# B&R Automation Studio project AriesV2 (part 3)

### bgsscanf.c
```c
#ifndef _BG_SSCANF_C
#define _BG_SSCANF_C
/*
Source:
http://www.koders.com/c/fid1D51E1E6F4F922088DF508FFEEEEC702AFED6333.aspx?s=__v_scanf
*/

//#include <stdarg.h>
//#include <limits.h>
//#include <string.h>

#define GBLONG_MAX 2147483647L
#define GBLONG_MIN (-GBLONG_MAX-1)
#define GBULONG_MAX (GBLONG_MAX * 2UL + 1)

extern long int strtol ( const char * str, char ** endptr, int base );

#define WANT_FLOATING_POINT_IN_SCANF 1
#define WANT_CHARACTER_CLASSES_IN_SCANF 1

#define	EOF	(-1)

struct arg_scanf {
  void *data;
  int (*getch)(void*);
  int (*putch)(int,void*);
};

struct str_data {
  unsigned char* str;
};

static int sgetc(struct str_data* sd) {
  register unsigned int ret = *(sd->str++);
  return (ret)?(int)ret:-1;
}

static int sputc(int c, struct str_data* sd) {
  return (*(--sd->str)==c)?c:-1;
}

#define A_GETC(fn)	(++consumed,(fn)->getch((fn)->data))
#define A_PUTC(c,fn)	(--consumed,(fn)->putch((c),(fn)->data))

static int isspace(int c)
{
	return ((c==(int)' ')) ? 1 : 0;
}

static int isdigit(int c)
{
	return ((c>=(int)'0') && (c<=(int)'9')) ? 1 : 0;
}

int __v_scanf(struct arg_scanf* fn, const unsigned char *format, va_list arg_ptr)
{
  unsigned int ch;	/* format act. char */
  int n=0;

  /* arg_ptr tmps */
#ifdef WANT_FLOATING_POINT_IN_SCANF
  double *pd;
  float  *pf;
#endif
  long   *pl;
  short  *ph;
  int    *pi;
  char    *s;

  unsigned int consumed=0;

  /* get one char */
  int tpch= A_GETC(fn);

  while (*format)
  {
    ch=*format++;
    switch (ch) {
    /* end of format string ?!? */
    case 0: return 0;

    /* skip spaces ... */
    case ' ':
    case '\f':
    case '\t':
    case '\v':
    case '\n':
    case '\r':
      while((*format)&&(isspace(*format))) ++format;
      while(isspace(tpch)) tpch=A_GETC(fn);
      break;

    /* format string ... */
    case '%':
      {
	unsigned int _div=0;
	int width=-1;
	char flag_width=0;
	char flag_discard=0;
	char flag_half=0;
	char flag_long=0;
	char flag_longlong=0;

in_scan:
	ch=*format++;
	if(ch!='n' && tpch==-1) goto err_out;
	switch (ch) {
	/* end of format string ?!? */
	case 0: return 0;

	/* check for % */
	case '%':
	  if ((unsigned char)tpch != ch) goto err_out;
	  tpch=A_GETC(fn);
	  break;

	/* FLAGS */
	case '*':
	  flag_discard=1;
	  goto in_scan;
	case 'h':
	  flag_half=1;
	  goto in_scan;
	case 'l':
	  if (flag_long) flag_longlong=1;
	  flag_long=1;
	  goto in_scan;
	case 'q':
	case 'L':
	  flag_longlong=1;
	  goto in_scan;

	/* WIDTH */
	case '0':
	case '1':
	case '2':
	case '3':
	case '4':
	case '5':
	case '6':
	case '7':
	case '8':
	case '9':
	  width=strtol((const char*)(format-1),&s,10);
	  format=(unsigned char*)s;
	  flag_width=1;
	  goto in_scan;

	/* scan for integer / strtol reimplementation ... */
	case 'p':
	case 'X':
	case 'x':
	  _div+=6;
	case 'd':
	  _div+=2;
	case 'o':
	  _div+=8;
	case 'u':
	case 'i':
	  {
	    unsigned long v=0;
	    unsigned int consumedsofar;
	    int neg=0;
	    while(isspace(tpch)) tpch=A_GETC(fn);
	    if (tpch=='-') {
	      tpch=A_GETC(fn);
	      neg=1;
	    }

	    if (tpch=='+') tpch=A_GETC(fn);

	    if (tpch==-1) return n;
	    consumedsofar=consumed;

	    if (!flag_width) {
	      if ((_div==16) && (tpch=='0')) goto scan_hex;
	      if (!_div) {
		_div=10;
		if (tpch=='0') {
		  _div=8;
scan_hex:
		  tpch=A_GETC(fn);
		  if ((tpch|32)=='x') {
		    tpch=A_GETC(fn);
		    _div=16;
		  }
		}
	      }
	    }
	    while ((width)&&(tpch!=-1)) {
	      register unsigned long c=tpch&0xff;
	      register unsigned long d=c|0x20;
	      c=(d>='a'?d-'a'+10:c<='9'?c-'0':0xff);
	      if (c>=_div) break;
	      d=v*_div;
	      v=(d<v)?GBULONG_MAX:d+c;
	      --width;
	      tpch=A_GETC(fn);
	    }

	    if (consumedsofar==consumed) return n;

	    if ((ch|0x20)<'p') {
	      register long l=v;
	      if (v>=-((unsigned long)GBLONG_MIN)) {
		l=(neg)?GBLONG_MIN:GBLONG_MAX;
	      }
	      else {
		if (neg) v*=-1;
	      }
	    }
	    if (!flag_discard) {
	      if (flag_long) {
		pl=(long *)va_arg(arg_ptr,long*);
		*pl=v;
	      } else if (flag_half) {
		ph=(short*)va_arg(arg_ptr,short*);
		*ph=v;
	      } else {
		pi=(int *)va_arg(arg_ptr,int*);
		*pi=v;
	      }
	      if(consumedsofar<consumed) ++n;
	    }
	  }
	  break;

	/* FIXME: return value of *scanf with ONE float maybe -1 instead of 0 */
#ifdef WANT_FLOATING_POINT_IN_SCANF
	/* floating point numbers */
	case 'e':
	case 'E':
	case 'f':
	case 'g':
	  {
	    double d=0.0;
	    int neg=0;
	    unsigned int consumedsofar;

	    while(isspace(tpch)) tpch=A_GETC(fn);

	    if (tpch=='-') {
	      tpch=A_GETC(fn);
	      neg=1;
	    }
	    if (tpch=='+') tpch=A_GETC(fn);

	    consumedsofar=consumed;

	    while (isdigit(tpch)) {
	      d=d*10+(tpch-'0');
	      tpch=A_GETC(fn);
	    }
	    if (tpch=='.') {
	      double factor=.1;
	      consumedsofar++;
	      tpch=A_GETC(fn);
	      while (isdigit(tpch)) {
		d=d+(factor*(tpch-'0'));
		factor/=10;
		tpch=A_GETC(fn);
	      }
	    }
	    if (consumedsofar==consumed) return n;	/* error */
	    if ((tpch|0x20)=='e') {
	      int exp=0, prec=tpch;
	      double factor=10;
	      tpch=A_GETC(fn);
	      if (tpch=='-') {
		factor=0.1;
		tpch=A_GETC(fn);
	      } else if (tpch=='+') {
		tpch=A_GETC(fn);
	      } else {
		d=0;
		if (tpch!=-1) A_PUTC(tpch,fn);
		tpch=prec;
		goto exp_out;
	      }
	      consumedsofar=consumed;
	      while (isdigit(tpch)) {
		exp=exp*10+(tpch-'0');
		tpch=A_GETC(fn);
	      }
	      if (consumedsofar==consumed) return n;	/* error */
	      while (exp) {	/* as in strtod: XXX: this introduces rounding errors */
		d*=factor; --exp;
	      }
	    }
exp_out:
	    if (!flag_discard) {
	      if (flag_long) {
		pd=(double *)va_arg(arg_ptr,double*);
		*pd=d;
	      } else {
		pf=(float *)va_arg(arg_ptr,float*);
		*pf=d;
	      }
	      ++n;
	    }
	  }
	  break;
#endif

	/* char-sequences */
	case 'c':
	  if (!flag_discard) {
	    s=(char *)va_arg(arg_ptr,char*);
	    ++n;
	  }
	  if (!flag_width) width=1;
	  while (width && (tpch!=-1)) {
	    if (!flag_discard) *(s++)=tpch;
	    --width;
	    tpch=A_GETC(fn);
	  }
	  break;

	/* string */
	case 's':
	  if (!flag_discard) s=(char *)va_arg(arg_ptr,char*);
	  while(isspace(tpch)) tpch=A_GETC(fn);
	  if (tpch==-1) break;		/* end of scan -> error */
	  while (width && (tpch!=-1) && (!isspace(tpch))) {
	    if (!flag_discard) *s=tpch;
	    if (tpch) ++s; else break;
	    --width;
	    tpch=A_GETC(fn);
	  }
	  if (!flag_discard) { *s=0; ++n; }
	  break;

	/* consumed-count */
	case 'n':
	  if (!flag_discard) {
	    pi=(int *)va_arg(arg_ptr,int *);
            *pi=consumed-1;
	  }
	  break;

#ifdef WANT_CHARACTER_CLASSES_IN_SCANF
	case '[':
	  {
	    char cset[256];
	    int flag_not=0;
	    int flag_dash=0;
	    memset(cset,0,sizeof(cset));
	    ch=*format++;
	    /* first char specials */
	    if (ch=='^') {
	      flag_not=1;
	      ch=*format++;
	    }
	    if ((ch=='-')||(ch==']')) {
	      cset[ch]=1;
	      ch=*format++;
	    }
	    /* almost all non special chars */
	    for (;(*format) && (*format!=']');++format) {
	      if (flag_dash) {
		register unsigned char tmp=*format;
		for (;ch<=tmp;++ch) cset[ch]=1;
		flag_dash=0;
		ch=*format;
	      }
	      else if (*format=='-') flag_dash=1;
	      else {
		cset[ch]=1;
		ch=*format;
	      }
	    }
	    /* last char specials */
	    if (flag_dash) cset['-']=1;
	    else cset[ch]=1;

	    /* like %c or %s */
	    if (!flag_discard) {
	      s=(char *)va_arg(arg_ptr,char*);
	      ++n;
	    }
	    while (width && (tpch>=0) && (cset[tpch]^flag_not)) {
	      if (!flag_discard) *s=tpch;
	      if (tpch) ++s; else break;
	      --width;
	      tpch=A_GETC(fn);
	    }
	    if (!flag_discard) *s=0;
	    ++format;
	  }
	  break;
#endif
	default:
	  goto err_out;
	}
      }
      break;

    /* check if equal format string... */
    default:
      if ((unsigned char)tpch != ch) goto err_out;
      tpch=A_GETC(fn);
      break;
    }
  }

  /* maybe a "%n" follows */
  if(*format) {
    while(isspace(*format)) format++;
    if(format[0] == '%' && format[1] == 'n') {
      pi = (int *) va_arg(arg_ptr, int *);
      *pi = consumed - 1;
    }
  }

err_out:
  if (tpch<0 && n==0) return EOF;
  A_PUTC(tpch,fn);
  return n;
}

int bgvsscanf(const char* str, const char* format, va_list arg_ptr)
{
  struct str_data  fdat = { (unsigned char*)str };
  struct arg_scanf farg = { (void*)&fdat, (int(*)(void*))sgetc, (int(*)(int,void*))sputc };
  return __v_scanf(&farg,format,arg_ptr);
}

int bgsscanf(const char *str, const char *format, ...)
{
  int n;
  va_list arg_ptr;
  va_start(arg_ptr, format);
  n=bgvsscanf(str,format,arg_ptr);
  va_end (arg_ptr);
  return n;
}

#endif
```

### bgTimer1ms.c
```c
/********************************************************************
 * COPYRIGHT -- belgor
 ********************************************************************
 * Package: bglib
 * File: bgTimer1ms.c
 * Author: goran
 * Created: October 05, 2011
 *******************************************************************/

#include <bur/plctypes.h>
#ifdef _DEFAULT_INCLUDES
	#include <AsDefault.h>
#endif

//#include <standard.h>

#ifndef _BG_TIMER_x1MS_C
#define _BG_TIMER_x1MS_C

void bgTimerExecute(TON_typ *timer){
	TON(timer);
}

void bgTimerStart(TON_typ *timer, int timeoutTime){
	timer->IN = 0;
	TON(timer);
	timer->IN = 1;
	timer->PT = timeoutTime;
	TON(timer );
}

void bgTimerStop(TON_typ *timer){
	timer->IN = 0;
	TON(timer);
}

BOOL  bgTimerIsTimeOut(TON_typ *timer){
	return timer->Q;
}

UDINT bgTimerTimeRemaining(TON_typ *timer){
	return (timer->PT - timer->ET);
}

UDINT bgTimerTimeElapsed( TON_typ *timer ) {
	return (timer->ET);
}

#endif //_BG_TIMER_x1MS_C
```

### HMI.typ
```iecst
(********************************************************************
 * COPYRIGHT -- piedmont
 ********************************************************************
 * Package: HMI
 * File: HMI.typ
 * Author: goran
 * Created: August 28, 2013
 ********************************************************************
 * Data types of package HMI
 ********************************************************************)
(*########################################################################*)
(*HMI key assinged PV-s (i.e. page navigation, save btns, etc)*)
(*########################################################################*)

TYPE
	hmiControlLogicKeys_typ : 	STRUCT
		btnRestartLoginTimer : USINT; (*1-means that login timer restart is requested*)
		btnLoginIcon : USINT; (*1-means that login logo (icon) is pressed*)
		menuKeyPressLT : ARRAY[0..HMI_ENUM_MENU_ITEMS_LT]OF BOOL; (*Mom keys connected to menu items LF*)
		menuKeyPressRT : ARRAY[0..HMI_ENUM_MENU_ITEMS_RT]OF BOOL; (*Mom keys connected to menu items RT*)
	END_STRUCT;
END_TYPE

(*########################################################################*)
(*HMI navigation PV-s (i.e. PV-s assigned to required VC PV-s such as currentPage, etc)*)
(*########################################################################*)

TYPE
	hmiNavigationLogic_typ : 	STRUCT
		changePage : USINT;
		currentPage : USINT;
		htmlCurrentURL : STRING[127];
		htmlChangeURL : STRING[127];
		currentPageText : STRING[31];
		prevPage : USINT;
		nextPage : USINT;
		pageInit : BOOL;
		pageExit : BOOL;
		state : USINT;
		currentStateText : STRING[31];
		statePrev : USINT;
		stateNext : USINT;
		loginLevel : UDINT;
		stateInit : BOOL;
		tmr1 : TON; (*Alert message control timer*)
		tmr2 : TON; (*Unack alarms message alert blinking timer*)
		tmr3 : TON; (*Password level reset timer*)
		tmr3RemainingTimeSec : UDINT;
		tmr3RemainingTimeMin : UDINT;
		tmr4 : TON;
	END_STRUCT;
END_TYPE

(*########################################################################*)
(*HMI related status control PV-s (i.e. visibility, locking, etc)*)
(*########################################################################*)

TYPE
	hmiControlLogicStatus_typ : 	STRUCT
		visibleSaveCfg : UINT;
		menuVisibleLT : UINT; (*Main menu LF visibility control *)
		menuVisibleRT : UINT; (*Main menu RT visibility control *)
		menuVisibleRTItems : ARRAY[0..HMI_ENUM_MENU_ITEMS_RT]OF UINT; (*Main menu items RT visibility control - for buttons stacked on top of each other in the upper, rt *)
		menuIndexLT : UINT; (*Main menu currently selected menu item - LF*)
		show_motion_tab : USINT;
		show_Aux_tab : USINT;
		show_io_tab : UINT;
		menuIndexRT : UINT; (*Main menu currently selected menu item - RT*)
		loginVisibleGE1 : USINT; (*Visibility control for login level related stuff - set to visible (0) if login level >= 1; othervise set to 1 (i.e. loginLevel < 1)*)
		loginVisibleGE2 : USINT; (*Visibility control for login level related stuff - set to visible (0) if login level >= 2; othervise set to 1 (i.e. loginLevel < 2)*)
		loginVisibleGE3 : USINT; (*Visibility control for login level related stuff - set to visible (0) if login level >= 2; othervise set to 1 (i.e. loginLevel < 2)*)
		menuLFHideTimer : TON; (*timer of automaticaly hiding LF dropdown menu*)
		menuRTHideTimer : TON; (*timer of automaticaly hiding RT dropdown menu*)
		tabKeysRadioDataPoint : USINT; (*DP that tab button are writing to in order to create radio buttons/tab view effect*)
		tabKeysRadioArray : ARRAY[0..HMI_ENUM_TAB_KEYS_MAX]OF USINT;
		tabKeysToggle : ARRAY[0..HMI_ENUM_MENU_ITEMS_LT]OF USINT;
		passwordStrings : ARRAY[0..HMI_PWD_LEVELS]OF STRING[HMI_PWD_MAXLEN]; (*Password strings used for loginLevel control*)
	END_STRUCT;
END_TYPE

(*=============================================================================*)
(*Recipe related HMI logic.*)
(*=============================================================================*)

TYPE
	hmiRecipeLogic_typ : 	STRUCT
		recVisible : USINT; (*Recipe related visibility control*)
		recSelectIdx : UINT; (*Recipe list index*)
		recSelectIdxMax : UINT; (*Recipe list index*)
		recSaveAsIdx : UINT; (*Recipe index for SaveAs action*)
		recSelectName : STRING[80]; (*Name of the currently selected recipe from the recipe list*)
		btnLockedActivate : USINT; (*Button lock control*)
		btnLockedNew : USINT; (*Button lock control*)
		btnLockedDelete : USINT; (*Button lock control*)
		btnLockedSaveAs : USINT; (*Button lock control*)
		btnActivate : BOOL; (*mom btn to Activate a recipe*)
		btnNew : BOOL; (*mom btn to New a recipe*)
		btnDelete : BOOL; (*mom btn to Delete a recipe*)
		btnSaveAs : BOOL; (*mom btn to SaveAs a recipe*)
		stateRecipes : UDINT;
	END_STRUCT;
END_TYPE

(*=============================================================================*)
(*Fileio Items*)
(*=============================================================================*)
(*=============================================================================*)
(*Tabs Control*)
(*=============================================================================*)
(*=============================================================================*)
(*HMI related navigation and control logic.*)
(*=============================================================================*)
(*Insert your comment here.*)
(*Insert your comment here.*)

TYPE
	hmiTableTrigger_typ : 	STRUCT
		Rec : BOOL;
		Cfg : BOOL;
	END_STRUCT;
	hmiTableLoad_typ : 	STRUCT
		Trigger : BOOL;
	END_STRUCT;
	hmiTables_typ : 	STRUCT
		Trigger : hmiTableTrigger_typ;
		Load : hmiTableLoad_typ;
	END_STRUCT;
END_TYPE

(*Insert your comment here.*)

TYPE
	hmiControlLogic_typ : 	STRUCT
		status : hmiControlLogicStatus_typ;
		keys : hmiControlLogicKeys_typ;
		prv : hmiNavigationLogic_typ; (*Hmi (panel) private data for handling screen navigation and hmi logic. Used only wihin HMI.*)
		recipes : hmiRecipeLogic_typ;
		alertMsg : hmiAlert_typ;
		dialogMsg : hmiDialog_typ;
		tables : hmiTables_typ;
	END_STRUCT;
END_TYPE
```

### HMI_Pages.typ
```iecst
TYPE
	HMI_Page_Enum :
		( (*IMPORTANTNOTE: if the application is going to work correctly, you have to MANUALLY ADD all of the enumerations below AND make sure they line up with the hmi page numbers. *)
		HMI_00_STARTUP := 0,
		HMI_HOME_10_DASHBOARD := 10,
		HMI_RECIPE_20_SELECT := 20,
		HMI_RECIPE_21_PVLIST := 21,
		HMI_CONFIG_30_SELECT := 30,
		HMI_CONFIG_31_PVLIST := 31,
		HMI_LOGIN_40_MAIN := 40,
		HMI_LOGIN_41_OPERATOR := 41,
		HMI_LOGIN_42_SETUP := 42,
		HMI_LOGIN_43_ENGINEER := 43,
		HMI_LOGIN_44_HERNON := 44,
		HMI_LOGIN_45_FACTORY := 45,
		HMI_DIAGNOSTICS_50_ALARMS := 50,
		HMI_DIAGNOSTICS_51_ALRMHST := 51,
		HMI_DIAGNOSTICS_52_SDM := 52,
		HMI_DIAGNOSTICS_53_SYSLOG := 53,
		HMI_MOTION_60_IO_DISPENSE := 60,
		HMI_MOTION_61_IO_MOTORS := 61,
		HMI_MOTION_62_DISPENSE_TREND := 62,
		HMI_MOTION_63_IO_INSPECT_IO := 63,
		HMI_MOTION_64_IO_INSPECT_TREND := 64,
		HMI_MOTION_65_IO_LOADER := 65,
		HMI_MOTION_66_IO_SAFETY := 66,
		HMI_MOTION_67_IO_ETC := 67,
		HMI_MOTION_68_IO_SENSOR := 68,
		HMI_MOTION_69_IO_LOAD5215 := 69,
		HMI_ACP_70_AXIS_OVERVIEW := 70,
		HMI_ACP_71_AXIS_REF := 71,
		HMI_ACP_72_AXIS_MOVE := 72,
		HMI_ACP_73_AXIS_SETUP := 73,
		HMI_ACP_74_CAM_CTRL := 74,
		HMI_ACP_75_CAM_SETUP := 75,
		HMI_ACP_76_CAM_TRACE := 76,
		HMI_AUX_90_FILE := 90
		);
END_TYPE
```

### HMIdialog.typ
```iecst
(********************************************************************
 * COPYRIGHT -- piedmont
 ********************************************************************
 * Package: HMI
 * File: HMI.typ
 * Author: goran
 * Created: August 28, 2013
 ********************************************************************
 * Data types of package HMI
 ********************************************************************)
(*########################################################################*)
(*HMI object - DIALOG (OK, Cancel)*)
(*########################################################################*)

TYPE
	hmiDialog_typ : 	STRUCT
		message : STRING[512];
		result : UINT; (*value returned when button pressed (0-busy, button not pressed, dialog active, OK pressed returns resultForOk (eg.1); Cancel pressed returns resultForCancel (eg.2)*)
		resultForOk : UINT; (*value to return when Ok pressed (if 0 return value is 1)*)
		resultForCancel : UINT; (*value to return when Cancel pressed (if 0 return value is 2)*)
		timeoutConfig : UINT; (*configuration input that defines meaning of the timeout. If 0 > timeout means cancel; if 1> timeout means ok*)
		status : UINT; (*Status for common dialog layer*)
		tmr1RemainingTimeSec : UDINT; (*Timer remaining time (sec)*)
		btnOk : UINT; (*press on button OK sets this value to 1*)
		btnCancel : UINT; (*press on button Cancel sets this value to 1*)
		tmr1 : TON; (*Dialog control timer*)
	END_STRUCT;
END_TYPE
```

### Program Logical/HMI/HMI_Alarms

#### Variables.var
```iecst
VAR
	ii_alarms : UDINT;
	tmp_alarm_counter : UDINT;
END_VAR
```

#### Cyclic.st
```iecst
PROGRAM _CYCLIC
	brsmemcpy(ADR(AppAlarms.AlarmImage[0]), 	ADR(gAlarms), 					SIZEOF(Machine_Alarms_typ));

	brsmemcpy(ADR(gAcknowledge), 				ADR(AppAlarms.AlarmImage[0]), 	SIZEOF(Machine_Alarms_typ));

//	tmp_alarm_counter := 0;
//
//	FOR ii_alarms := 0 TO MAX_IDX_ALARMS BY 1 DO
//		IF gMachine.HMI.AlarmControls.Dispense.AlarmImage[ii_alarms] THEN
//			tmp_alarm_counter := tmp_alarm_counter + 1;
//		END_IF;
//
//		IF gMachine.HMI.AlarmControls.Inspect.AlarmImage[ii_alarms] THEN
//			tmp_alarm_counter := tmp_alarm_counter + 1;
//		END_IF;
//
//		IF gMachine.HMI.AlarmControls.Sensor.AlarmImage[ii_alarms] THEN
//			tmp_alarm_counter := tmp_alarm_counter + 1;
//		END_IF;
//
//		IF gMachine.HMI.AlarmControls.Safety.AlarmImage[ii_alarms] THEN
//			tmp_alarm_counter := tmp_alarm_counter + 1;
//		END_IF;
//
//		IF gMachine.HMI.AlarmControls.RecCfg.AlarmImage[ii_alarms] THEN
//			tmp_alarm_counter := tmp_alarm_counter + 1;
//		END_IF;
//
//		IF gMachine.HMI.AlarmControls.Hardware.AlarmImage[ii_alarms] THEN
//			tmp_alarm_counter := tmp_alarm_counter + 1;
//		END_IF;
//
//		IF gMachine.HMI.AlarmControls.Motor.AlarmImage[ii_alarms] THEN
//			tmp_alarm_counter := tmp_alarm_counter + 1;
//		END_IF;
//	END_FOR;

	IF gAlarmResetRequested THEN
		brsmemset(ADR(gAlarms), 0, 		SIZEOF(Machine_Alarms_typ));

		gAlarmResetRequested := FALSE;
	END_IF;
//
//	IF Alarm_Control.ActiveAlarms = 0 AND Alarm_Control.PendingAlarms = 0 AND tmp_alarm_counter = 0 THEN
//		gAlarmState := 0;
//	ELSIF Alarm_Control.ActiveAlarms = 0 AND Alarm_Control.PendingAlarms = 0 AND tmp_alarm_counter > 0 THEN
//		gAlarmState := 1;
//	ELSIF Alarm_Control.ActiveAlarms = 0 AND Alarm_Control.PendingAlarms > 0 THEN
//		gAlarmState := 2;
//	ELSE
//		gAlarmState := 3;
//	END_IF;

	AppAlarms_FBK();
//
//	gMachine.HMI.Dashboard.Application_Errors_Active := tmp_alarm_counter;
//	gMachine.HMI.Dashboard.System_Alarms_Active := Alarm_Control.ActiveAlarms;
//	gMachine.HMI.Dashboard.System_Alarms_Pending := Alarm_Control.PendingAlarms;
END_PROGRAM
```

### Program Logical/HMI/hmilogic

#### hmiDialog.h
```c
/********************************************************************
 * COPYRIGHT -- piedmont
 ********************************************************************
 * Program: hmilogic
 * File: hmiDialog.h
 * Author: goran
 * Created: September 05, 2013
 *******************************************************************/

#include <bur/plctypes.h>
#ifdef _DEFAULT_INCLUDES
#include <AsDefault.h>
#endif
BOOL hmiDialogIsActive(hmiDialog_typ* p);
void hmiDialogHide(hmiDialog_typ* p);
void hmiDialogShow(hmiDialog_typ* p, char* msg, UINT timeout_ms, UINT resultForOk, UINT resultForCancel, UINT timeoutConfig);
UINT hmiDialogCyclic(hmiDialog_typ* p);
```

#### loginCyclicLogic.c
```c
#include <bur/plctypes.h>
#ifdef _DEFAULT_INCLUDES
#include <AsDefault.h>
#endif

void loginLevelParameterEditControl(UDINT minLevel)
{
	//input form (i.e. common page) not visible for operator
	//(i.e. loginlevel==0 > visibility set to 1 (not visible))
	/*gHmiParamTable.selValueFormVisible = (gHmi.prv.loginLevel >= minLevel) ? 0 : 1;*/
	gHmiParamTable.selValueFormVisible = 0;
}

//login level related logic
void	loginLevelLogicCyclic()
{
	static UINT loginLevelOld;

	//update visiblity flags that are associated with the current login level
	//note that current app support three login levels: 0-operator;1-supervisor;2-admin
//	if(gHmi.prv.loginLevel == 1){
//		gHmi.status.loginVisibleGE1 = 0;//visible
//		gHmi.status.loginVisibleGE2 = 1;//not visible
//		gHmi.status.loginVisibleGE3 = 1;//not visible
//	}else
//		if(gHmi.prv.loginLevel == 2){
//		gHmi.status.loginVisibleGE1 = 0;//visible
//		gHmi.status.loginVisibleGE2 = 0;//visible
//		gHmi.status.loginVisibleGE3 = 1;//not visible
//	}else
//		if(gHmi.prv.loginLevel == 3){
//		gHmi.status.loginVisibleGE1 = 0;//visible
//		gHmi.status.loginVisibleGE2 = 0;//visible
//		gHmi.status.loginVisibleGE3 = 0;//visible
//	}else{
//		gHmi.status.loginVisibleGE1 = 1;//not visible
//		gHmi.status.loginVisibleGE2 = 1;//not visible
//		gHmi.status.loginVisibleGE3 = 1;//not visible
//	}

	gHmi.status.loginVisibleGE1 = 0;//visible
	gHmi.status.loginVisibleGE2 = 0;//visible
	gHmi.status.loginVisibleGE3 = 0;//visible

	//operate login timeout timer
	//Timer for timed out operation of the access control

	bgTimerCyclic(&gHmi.prv.tmr3) ;

	//detect login level changes
	if(gHmi.prv.loginLevel != loginLevelOld){
		loginLevelOld = gHmi.prv.loginLevel;
		if(gHmi.prv.loginLevel){
			//when supervisor or admin logs in > start login timeout timer
			bgTimerStart(&gHmi.prv.tmr3, Tms(DEFINE_LOGIN_TO)); //login duration timer setting comes from current config [sec], convert to [ms]
		}else{
			//when loginLevel gets reset to 0, make sure to make the parametar input field invisible
			loginLevelParameterEditControl(1);
		}
	}

	//restart login timer if user touches the area of the ticking logout timer
	if(gHmi.keys.btnRestartLoginTimer){
		gHmi.keys.btnRestartLoginTimer = 0;
		bgTimerStart(&gHmi.prv.tmr3, Tms(DEFINE_LOGIN_TO));
	}

	//change page to login is user touches the area of the login icon
	if(gHmi.keys.btnLoginIcon){
		gHmi.keys.btnLoginIcon = 0;
		if(!gHmi.prv.loginLevel){
			gHmi.prv.changePage = HMI_LOGIN_40_MAIN;
		}
	}

	//timer based logout > if loginLeve higher then 0, reset it after timer expires
	if(gHmi.prv.loginLevel && bgTimerIsTimeOut(&gHmi.prv.tmr3)){
		gHmi.prv.loginLevel = 0;
	}

	//calculate remaining login time [min:sec] from remaining timer time [ms]
	gHmi.prv.tmr3RemainingTimeSec = (bgTimerTimeRemaining(&gHmi.prv.tmr3)/1000) % 60;
	gHmi.prv.tmr3RemainingTimeMin = (bgTimerTimeRemaining(&gHmi.prv.tmr3)/1000) / 60;

}
```

### Program Logical/HMI/HMITableManager (IEC)

#### Main.st - Init, cyclic, exit code
```iecst
PROGRAM _INIT
	//loadHMITable is a FBK with structures containing the values loaded from the textsystem files
	loadHMITable[TABLE_RECIPE]		(tableName := 'Process Recipe',			nameSpace := 'hmiTable/Recipe',	Logbook := Init_Logbook.pLog, 	pOverallStats := ADR(tableStats.Overall));
	loadHMITable[TABLE_CONFIG]		(tableName := 'Machine Configuration',	nameSpace := 'hmiTable/Config',	Logbook := Init_Logbook.pLog, 	pOverallStats := ADR(tableStats.Overall));
END_PROGRAM

//TODO: Load param array with %s, replace with index.
//TODO: More scrutiny to ensure tables were done correctly

PROGRAM _CYCLIC
	IF gHmi.tables.Trigger.Rec THEN
		gHmi.tables.Trigger.Rec := FALSE;
		ActivateHMITable(gRecCfg.active.Cfg.HMI.MachineLang, pHMITable := ADR(gHmiParamTable), pTableValues := ADR(loadHMITable[TABLE_RECIPE].hmiStruct));//No Control recipe values
	END_IF;

	IF gHmi.tables.Trigger.Cfg THEN
		gHmi.tables.Trigger.Cfg := FALSE;
		ActivateHMITable(gRecCfg.active.Cfg.HMI.MachineLang, pHMITable := ADR(gHmiParamTable), pTableValues := ADR(loadHMITable[TABLE_CONFIG].hmiStruct));//No Control recipe values
	END_IF;

	hmiParamListTableCyclic(ADR(gHmiParamTable));

END_PROGRAM
```

- Data object Logical/acp10etxen (Ett) (no source held here)

- Data object Logical/Axisobj/Axisi (Ax) (no source held here)

- Program Logical/MotionControl/LineControl (IEC) - Manage all ACP10, MpAxis functionality for the line control (no source held here)

Listed in the project but not available here: Logical/Libraries/jgLibC/Types.typ, Logical/Libraries/jgLibC/Constants.var, Logical/Libraries/jgLibC/jgLibC.fun, Logical/Libraries/jgLibC/Debounce_Signal.c, Logical/Libraries/wbrServices/TimerServices/TimerServices.typ, Logical/Libraries/wbrServices/TimerServices/msTimeSvc/msTimeSvc.c, Logical/Libraries/wbrServices/wbrMemSvc/wbrMemSvc.fun, Logical/Libraries/wbrServices/wbrMemSvc/wbrMemSvc.c, Logical/Libraries/wbrServices/wbrPingSvc/wbrPingSvc.typ, Logical/Libraries/wbrServices/wbrPingSvc/wbrPingSvc.fun, Logical/Libraries/wbrServices/wbrPingSvc/wbrPingSvc.c, Logical/Libraries/wbrServices/wbrsprintf/wbrsprintf.h, Logical/Libraries/wbrServices/wbrsprintf/cvtflasc.c, Logical/Libraries/wbrServices/wbrSvcUtilities/wbrFltUtil/wbrFltUtil.fun, Logical/Libraries/wbrServices/wbrSvcUtilities/wbrFltUtil/wbrFloatUtilities.c, Logical/HMI/HMITableManager/Types.typ, Logical/HMI/HMITableManager/Variables.var, Logical/MotionControl/MotionVar.var, Logical/MotionControl/LineControl/Main.st, Logical/MotionControl/LineControl/Types.typ, Logical/MotionControl/LineControl/Variables.var
